{region '#Template'}
	{attribute 'Category' := 'GVLs'}
	{attribute 'Version' := '0.0.1.0'}
	{attribute 'Tags' := 'DPAD, Trades, ObjectName, Description'}
	{attribute 'Description' := 'Textliste Gewerke	// Text list trades'}
{endregion}
{attribute 'qualified_only'}
VAR_GLOBAL
  Doors_gates_windows_sun_protection_sObjectName                :T_MaxString:= 'TTF';
  Doors_gates_windows_sun_protection_sDescription               :T_MaxString:= 'Türen, Tore, Fenster, Sonnenschutz';
  Sewage_water_and_gas_plants_sObjectName                       :T_MaxString:= 'GWA';
  Sewage_water_and_gas_plants_sDescription                      :T_MaxString:= 'Abwasser-, Wasser-, Gasanlagen';
  Heat_supply_systems_sObjectName                               :T_MaxString:= 'HZG';
  Heat_supply_systems_sDescription                              :T_MaxString:= 'Wärmeversorgungsanlagen';
  Ventilation_systems_sDescription                              :T_MaxString:= 'Lufttechnische Anlagen';
  Ventilation_systems_sObjectName                               :T_MaxString:= 'RLT';
  Refrigeration_systems_sObjectName                             :T_MaxString:= 'KAE';
  Refrigeration_systems_sDescription                            :T_MaxString:= 'Kälteanlagen';
  High_voltage_systems_sObjectName                              :T_MaxString:= 'ELT';
  High_voltage_systems_sDescription                             :T_MaxString:= 'Starkstromanlagen';
  Telecommunication_and_information_technology_sObjectName      :T_MaxString:= 'FIA';
  Telecommunication_and_information_technology_sDescription     :T_MaxString:= 'Fernmelde- und informationstechnische Anlagen';
  Hazard_detection_and_alarm_systems_sObjectName                :T_MaxString:= 'GMA';
  Hazard_detection_and_alarm_systems_sDescription               :T_MaxString:= 'Gefahrenmelde- und Alarmanlagen';
  Conveyors_sObjectName                                         :T_MaxString:= 'FTA';
  Conveyors_sDescription                                        :T_MaxString:= 'Förderanlagen';
  Kitchen_technology_systems_sObjectName                        :T_MaxString:= 'KTA';
  Kitchen_technology_systems_sDescription                       :T_MaxString:= 'Küchentechnische Anlagen';
  Laundry_and_cleaning_systems_sObjectName                      :T_MaxString:= 'WRA';
  Laundry_and_cleaning_systems_sDescription                     :T_MaxString:= 'Wäscherei- und Reinigungsanlagen';
  Media_supply_systems_sObjectName                              :T_MaxString:= 'MVA';
  Media_supply_systems_sDescription                             :T_MaxString:= 'Medienversorgungsanlagen';
  Medical_and_laboratory_equipment_sObjectName                  :T_MaxString:= 'MED';
  Medical_and_laboratory_equipment_sDescription                 :T_MaxString:= 'Medizin- und labortechnische Anlagen';
  Fire_extinguishing_systems_sObjectName                        :T_MaxString:= 'FLA';
  Fire_extinguishing_systems_sDescription                       :T_MaxString:= 'Feuerlöschanlagen';
  Bathing_facilities_sObjectName                                :T_MaxString:= 'BTA';
  Bathing_facilities_sDescription                               :T_MaxString:= 'Badetechnische Anlagen';
  Process_heating_cooling_and_air_systems_sObjectName           :T_MaxString:= 'PRO';
  Process_heating_cooling_and_air_systems_sDescription          :T_MaxString:= 'Prozesswärme-, -kälte- und -luftanlagen';
  Waste_disposal_facilities_sObjectName                         :T_MaxString:= 'ENT';
  Waste_disposal_facilities_sDescription                        :T_MaxString:= 'Entsorgungsanlagen';
  Building_automation_and_control_systems_general_sObjectName   :T_MaxString:= 'GAS';
  Building_automation_and_control_systems_general_sDescription  :T_MaxString:= 'Gebäudeautomation allgemein';
  Automation_focal_point_information_focal_point_sObjectName    :T_MaxString:= 'ISP';
  Automation_focal_point_information_focal_point_sDescription   :T_MaxString:= 'Automationsschwerpunkt/Informationsschwerpunkt';
  Room_automation_sObjectName                                   :T_MaxString:= 'RAU';
  Room_automation_sDescription                                  :T_MaxString:= 'Raumautomation';
  Technical_equipment_in_outdoor_facilities_sObjectName         :T_MaxString:= 'TAA';
  Technical_equipment_in_outdoor_facilities_sDescription        :T_MaxString:= 'Technische Anlagen in Außenanlagen';
	
END_VAR

(* stored: Version 1.1.0.1, ProductVersion 3.1.4024.6
   GVL TextTrades: Id {de9d6cee-08be-4e79-961e-3f37ba4360b7} *)
